RoboDK station: Example 3 - Unload pallet.rdk

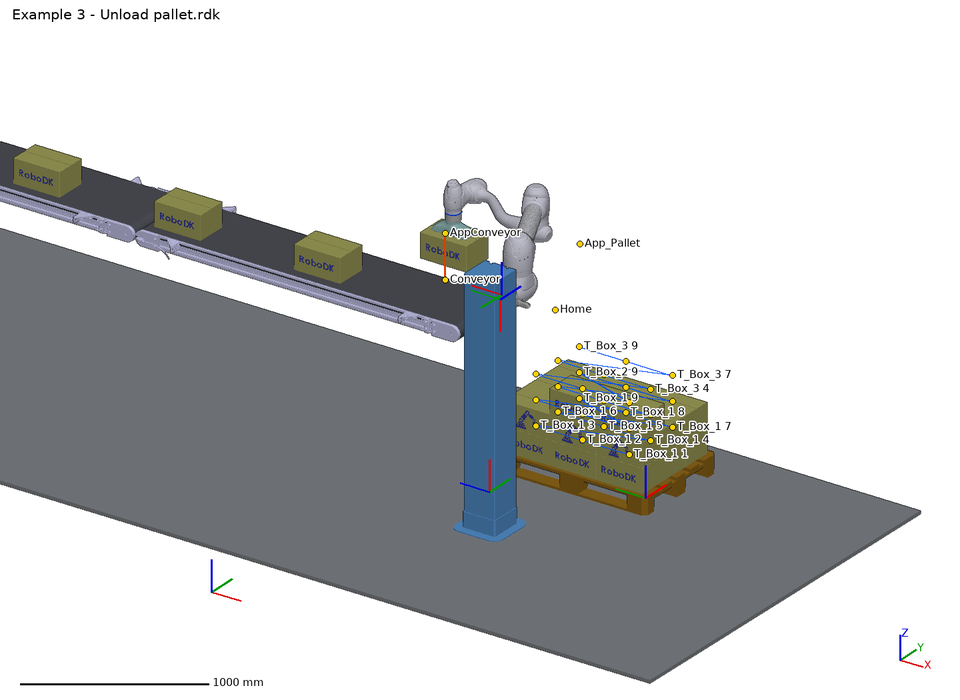
[picture v0: the station drawn from its stored meshes, robots at their saved joint values, targets as dots, program paths as lines]
Station Example 3 - Unload pallet. Poses are relative to the parent item; angles as X-Y-Z fixed-axis rotations.
  - frame Linear Rail Base at (750, 1500, 200) mm, rotated rx 0 ry -90 rz 0 deg
    - robot Linear Rail: 1 axes
        modified DH rows (alpha deg, a mm, theta deg, d mm): 0, 0, 0, 0 linear
        base shift (0, 0, 0) mm, rotated rx 0 ry 90 rz 0 deg
        joint limits [0] to [1200]; home [0]; saved at [1095.81]
      - frame Doosan Robotics M1013 Base at (0, 100, 0) mm, rotated rx 90 ry 0 rz 180 deg
        - robot Doosan Robotics M1013: 6 axes, payload 10 kg, reach 1300 mm, repeatability 0.1 mm, weight 33 kg
            modified DH rows (alpha deg, a mm, theta deg, d mm): 0, 0, 0, 152.5; -90, 0, -90, 34.506; 0, 620, -90, 0; -90, 0, 0, 559; 90, 0, 0, 0; -90, 0, 180, 121
            base shift (0, 0, 0) mm, rotated rx 0 ry 0 rz 180 deg
            joint limits [-120, -100, -160, -360, -360, -360] to [-60, 100, 160, 360, 360, 360]; home [0, 0, -90, 0, 0, 0]; saved at [-88.555, 26.122, 60.089, 89.791, -91.38, -93.79]
          - tool Tool, TCP at (0, 0, 69) mm, size 225 x 100 x 69 mm, geometry from Tool.step
            - object Box_3 3 at (5, 0, 77.5) mm, rotated rx 180 ry 0 rz -90 deg, size 300 x 202 x 153 mm, geometry from Box.step
  - frame Conveyor Belt Base at (57.17, 2600, 730) mm, rotated rx 0 ry 0 rz -180 deg
    - robot Conveyor Belt: 1 axes
        modified DH rows (alpha deg, a mm, theta deg, d mm): 0, 0, 0, 0 linear
        base shift (0, 0, 0) mm, rotated rx 0 ry 90 rz 0 deg
        joint limits [-500000] to [500000]; home [0]; saved at [-494045.004]
      - frame Conveyor at (0, 0, 0) mm
        - object Box_3 9 at (499511.41, 284.96, 74.77) mm, rotated rx 0.03 ry -0.02 rz -90.02 deg, size 300 x 202 x 153 mm, geometry from Box.step
        - object Box_3 8 at (498601.41, 284.96, 74.77) mm, rotated rx 0.03 ry -0.02 rz -90.02 deg, size 300 x 202 x 153 mm, geometry from Box.step
        - object Box_3 7 at (497699.41, 284.96, 74.77) mm, rotated rx 0.03 ry -0.02 rz -90.02 deg, size 300 x 202 x 153 mm, geometry from Box.step
        - object Box_3 6 at (496784.41, 284.96, 74.77) mm, rotated rx 0.03 ry -0.02 rz -90.02 deg, size 300 x 202 x 153 mm, geometry from Box.step
        - object Box_3 5 at (495873.41, 284.96, 74.77) mm, rotated rx 0.03 ry -0.02 rz -90.02 deg, size 300 x 202 x 153 mm, geometry from Box.step
        - object Box_3 4 at (494970.41, 284.96, 74.77) mm, rotated rx 0.03 ry -0.02 rz -90.02 deg, size 300 x 202 x 153 mm, geometry from Box.step
    - target AppConveyor (Cartesian target) at (166.39, 285.12, 428.8) mm, rotated rx -179.99 ry 0.02 rz 179.99 deg; joints [-88.768, 29.095, 58.796, 89.941, -91.212, -92.104, 1095.81] of Doosan Robotics M1013
    - target Conveyor (Cartesian target) at (166.37, 284.98, 152.27) mm, rotated rx -179.98 ry 0.03 rz 179.98 deg; joints [-88.76, 29.09, 58.79, 89.94, -91.21, -92.1, 819.16] of Doosan Robotics M1013
    - object Conveyor at (2400, 440, -50) mm, rotated rx 0 ry 0 rz -90 deg, size 597 x 2090.8 x 107.2 mm
    - object Conveyor at (4500, 440, -50) mm, rotated rx 0 ry 0 rz -90 deg, size 597 x 2090.8 x 107.2 mm
  - frame Pallet at (1350, 2080, 100) mm, rotated rx 0 ry 0 rz 90 deg
    - object Pallet at (-0.19, 0.17, 1.21) mm, size 660 x 990 x 118.8 mm, geometry from User Library-Europallet.igs
    - target T_Box_1 1 (Cartesian target) at (120, 190, 157.5) mm, rotated rx -180 ry 0 rz -90 deg; joints [-92.925, -96.78, 118.114, 92.725, -88.936, -158.691, 192] of Doosan Robotics M1013
    - target T_Box_1 2 (Cartesian target) at (120, 490, 157.5) mm, rotated rx 180 ry 0 rz -90 deg; joints [-100.509, -74.899, 134.13, 95.421, -80.984, -121.197, 192] of Doosan Robotics M1013
    - target T_Box_1 3 (Cartesian target) at (120, 790, 157.5) mm, rotated rx 180 ry 0 rz -90 deg; joints [-83.756, -35.637, 131.426, 90.632, -96.212, -84.176, 192] of Doosan Robotics M1013
    - target T_Box_1 4 (Cartesian target) at (320, 190, 157.5) mm, rotated rx -180 ry 0 rz -90 deg; joints [-92.925, -78.491, 98.933, 92.741, -88.979, -159.582, 192] of Doosan Robotics M1013
    - target T_Box_1 5 (Cartesian target) at (320, 490, 157.5) mm, rotated rx -180 ry 0 rz -90 deg; joints [-100.509, -62.114, 112.355, 96.766, -81.94, -130.236, 192] of Doosan Robotics M1013
    - target T_Box_1 6 (Cartesian target) at (320, 790, 157.5) mm, rotated rx 180 ry 0 rz -90 deg; joints [-83.756, -34.116, 110.225, 88.495, -96.061, -103.971, 192] of Doosan Robotics M1013
    - target T_Box_1 7 (Cartesian target) at (520, 190, 157.5) mm, rotated rx 180 ry 0 rz -90 deg; joints [-92.925, -60.698, 73.974, 92.847, -89.329, -166.74, 192] of Doosan Robotics M1013
    - target T_Box_1 8 (Cartesian target) at (520, 490, 157.5) mm, rotated rx 180 ry 0 rz -90 deg; joints [-100.509, -48.668, 87.076, 98.271, -83.494, -142.063, 192] of Doosan Robotics M1013
    - target T_Box_1 9 (Cartesian target) at (520, 790, 157.5) mm, rotated rx 180 ry 0 rz -90 deg; joints [-83.756, -26.873, 85.087, 86.702, -95.305, -121.939, 192] of Doosan Robotics M1013
    - target T_Box_2 1 (Cartesian target) at (120, 190, 310) mm, rotated rx -180 ry 0 rz -90 deg; joints [-100, -10.355, 75.202, 134.117, -34.001, -139.471, 347.5] of Doosan Robotics M1013
    - target T_Box_2 2 (Cartesian target) at (120, 490, 310) mm, rotated rx 180 ry 0 rz -90 deg; joints [-100, -10.355, 75.202, 134.117, -34.001, -139.471, 347.5] of Doosan Robotics M1013
    - target T_Box_2 3 (Cartesian target) at (120, 790, 310) mm, rotated rx 180 ry 0 rz -90 deg; joints [-100, -10.355, 75.202, 134.117, -34.001, -139.471, 347.5] of Doosan Robotics M1013
    - target T_Box_2 4 (Cartesian target) at (320, 190, 310) mm, rotated rx -180 ry 0 rz -90 deg; joints [-100, -10.355, 75.202, 134.117, -34.001, -139.471, 347.5] of Doosan Robotics M1013
    - target T_Box_2 5 (Cartesian target) at (320, 490, 310) mm, rotated rx -180 ry 0 rz -90 deg; joints [-100, -10.355, 75.202, 134.117, -34.001, -139.471, 347.5] of Doosan Robotics M1013
    - target T_Box_2 6 (Cartesian target) at (320, 790, 310) mm, rotated rx 180 ry 0 rz -90 deg; joints [-100, -10.355, 75.202, 134.117, -34.001, -139.471, 347.5] of Doosan Robotics M1013
    - target T_Box_2 7 (Cartesian target) at (520, 190, 310) mm, rotated rx 180 ry 0 rz -90 deg; joints [-100, -10.355, 75.202, 134.117, -34.001, -139.471, 347.5] of Doosan Robotics M1013
    - target T_Box_2 8 (Cartesian target) at (520, 490, 310) mm, rotated rx 180 ry 0 rz -90 deg; joints [-100, -10.355, 75.202, 134.117, -34.001, -139.471, 347.5] of Doosan Robotics M1013
    - target T_Box_2 9 (Cartesian target) at (520, 790, 310) mm, rotated rx 180 ry 0 rz -90 deg; joints [-100, -10.355, 75.202, 134.117, -34.001, -139.471, 347.5] of Doosan Robotics M1013
    - target T_Box_3 1 (Cartesian target) at (120, 190, 462.5) mm, rotated rx -180 ry 0 rz -90 deg; joints [-92.508, -96.765, 118.144, 92.336, -89.086, -158.639, 500] of Doosan Robotics M1013
    - target T_Box_3 2 (Cartesian target) at (120, 490, 462.5) mm, rotated rx 180 ry 0 rz -90 deg; joints [-99.069, -74.746, 134.167, 94.642, -82.201, -120.896, 500] of Doosan Robotics M1013
    - target T_Box_3 3 (Cartesian target) at (120, 790, 462.5) mm, rotated rx 180 ry 0 rz -90 deg; joints [-84.635, -35.739, 131.462, 90.537, -95.338, -84.252, 500] of Doosan Robotics M1013
    - target T_Box_3 4 (Cartesian target) at (320, 190, 462.5) mm, rotated rx -180 ry 0 rz -90 deg; joints [-92.508, -78.478, 98.96, 92.35, -89.123, -159.536, 500] of Doosan Robotics M1013
    - target T_Box_3 5 (Cartesian target) at (320, 490, 462.5) mm, rotated rx -180 ry 0 rz -90 deg; joints [-99.069, -62.008, 112.384, 95.812, -83.027, -129.979, 500] of Doosan Robotics M1013
    - target T_Box_3 6 (Cartesian target) at (320, 790, 462.5) mm, rotated rx 180 ry 0 rz -90 deg; joints [-84.635, -34.196, 110.254, 88.704, -95.206, -104.001, 500] of Doosan Robotics M1013
    - target T_Box_3 7 (Cartesian target) at (520, 190, 462.5) mm, rotated rx 180 ry 0 rz -90 deg; joints [-92.508, -60.689, 74.002, 92.441, -89.423, -166.699, 500] of Doosan Robotics M1013
    - target T_Box_3 8 (Cartesian target) at (520, 490, 462.5) mm, rotated rx 180 ry 0 rz -90 deg; joints [-99.069, -48.589, 87.102, 97.119, -84.367, -141.837, 500] of Doosan Robotics M1013
    - target T_Box_3 9 (Cartesian target) at (520, 790, 462.5) mm, rotated rx 180 ry 0 rz -90 deg; joints [-100, -10.355, 75.202, 134.117, -34.001, -139.471, 500] of Doosan Robotics M1013
    - target App_Pallet (Cartesian target) at (536.24, 799.31, 1058.38) mm, rotated rx -179.99 ry 0.02 rz -90.01 deg; joints [-84.86, -25.42, 82.51, 87.2, -94.29, -123.01, 1095.81] of Doosan Robotics M1013
    - object Box_1 1 at (120, 185, 80) mm, size 300 x 202 x 153 mm, geometry from Box.step
    - object Box_1 2 at (120, 485, 80) mm, size 300 x 202 x 153 mm, geometry from Box.step
    - object Box_1 3 at (120, 785, 80) mm, size 300 x 202 x 153 mm, geometry from Box.step
    - object Box_1 4 at (320, 185, 80) mm, size 300 x 202 x 153 mm, geometry from Box.step
    - object Box_1 5 at (320, 485, 80) mm, size 300 x 202 x 153 mm, geometry from Box.step
    - object Box_1 6 at (320, 785, 80) mm, size 300 x 202 x 153 mm, geometry from Box.step
    - object Box_1 7 at (520, 185, 80) mm, size 300 x 202 x 153 mm, geometry from Box.step
    - object Box_1 8 at (520, 485, 80) mm, size 300 x 202 x 153 mm, geometry from Box.step
    - object Box_1 9 at (520, 785, 80) mm, size 300 x 202 x 153 mm, geometry from Box.step
    - object Box_2 1 at (520, 785, 232.5) mm, rotated rx 0 ry 0 rz -180 deg, size 300 x 202 x 153 mm, geometry from Box.step
    - object Box_2 2 at (520, 485, 232.5) mm, rotated rx 0 ry 0 rz -180 deg, size 300 x 202 x 153 mm, geometry from Box.step
    - object Box_2 3 at (520, 185, 232.5) mm, rotated rx 0 ry 0 rz -180 deg, size 300 x 202 x 153 mm, geometry from Box.step
    - object Box_2 4 at (320, 785, 232.5) mm, rotated rx 0 ry 0 rz -180 deg, size 300 x 202 x 153 mm, geometry from Box.step
    - object Box_2 5 at (320, 485, 232.5) mm, rotated rx 0 ry 0 rz -180 deg, size 300 x 202 x 153 mm, geometry from Box.step
    - object Box_2 6 at (320, 185, 232.5) mm, rotated rx 0 ry 0 rz -180 deg, size 300 x 202 x 153 mm, geometry from Box.step
    - object Box_2 7 at (120, 785, 232.5) mm, rotated rx 0 ry 0 rz -180 deg, size 300 x 202 x 153 mm, geometry from Box.step
    - object Box_2 8 at (120, 485, 232.5) mm, rotated rx 0 ry 0 rz -180 deg, size 300 x 202 x 153 mm, geometry from Box.step
    - object Box_2 9 at (120, 185, 232.5) mm, rotated rx 0 ry 0 rz -180 deg, size 300 x 202 x 153 mm, geometry from Box.step
    - object Box_3 1 at (120, 185, 385) mm, size 300 x 202 x 153 mm, geometry from Box.step
    - object Box_3 2 at (120, 485, 385) mm, size 300 x 202 x 153 mm, geometry from Box.step
  - frame World at (0, 0, 0) mm
    - target Home (joint target) at (876.47, 1924.34, 1140.31) mm, rotated rx -180 ry 0 rz 0 deg; joints [-90, -100, 160, 90, -90, -120, 1095.8] of Doosan Robotics M1013
    - target ConvHome (Cartesian target) at (500057.17, 2600, 730) mm, rotated rx 0 ry 0 rz -180 deg; joints [-500000, 0, 0, 0, 0, 0, 0] of Conveyor Belt
    - target ConvRun (Cartesian target) at (392.51, 2433.37, 999.75) mm, rotated rx 180 ry 0 rz 2.38 deg; joints [50000, -58.983, -101.068, -19.936, -5.281, -2.394, 1150.26] of Conveyor Belt
    - object Floor at (-7500, 480, -30) mm, size 10000 x 2500 x 20 mm, geometry from Floor.step
  - program ReplaceObjects (1 instructions, listed below)
  - program MainProgram (167 instructions, listed below)
  - program AppPallet (3 instructions, listed below)
  - program DropConveyor (6 instructions, listed below)
  - program GoHome (3 instructions, listed below)
  - program Pick (1 instructions, listed below)
  - program RunConveyor (2 instructions, listed below)
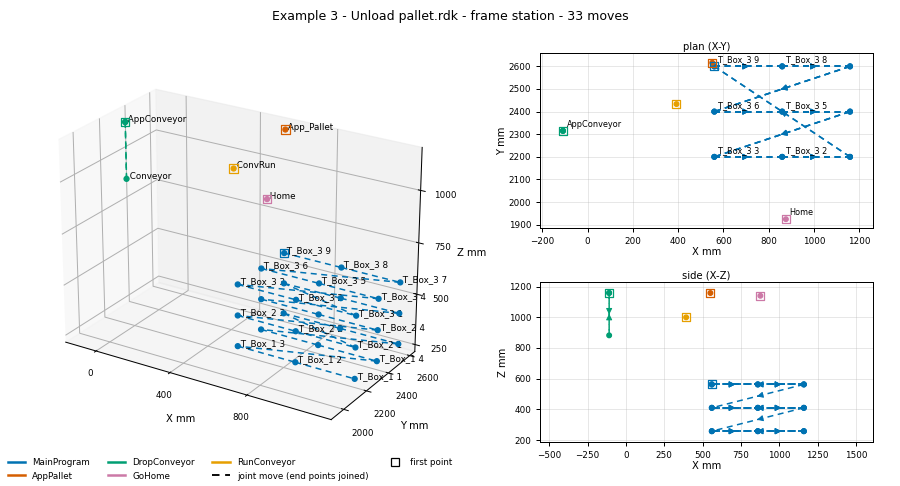
[picture p0: tool path of Example 3 - Unload pallet.rdk in frame station, 33 of 33 moves have a stored position in this frame; points joined in program order, loops and branches not executed]

--- program ReplaceObjects (robot Doosan Robotics M1013) ---
  Replace objects

--- program MainProgram (robot Doosan Robotics M1013) ---
  Call GoHome
  Call ReplaceObjects
  Pause 10.0 s
  Run RunConveyor
  Set Ref.: Pallet
  MoveJ (T_Box_3 9)
  Call Pick
  Call AppPallet
  Call DropConveyor
  Call AppPallet
  Set Ref.: Pallet
  MoveJ (T_Box_3 8)
  Call Pick
  Call AppPallet
  Call DropConveyor
  Call AppPallet
  Set Ref.: Pallet
  MoveJ (T_Box_3 7)
  Call Pick
  Call AppPallet
  Call DropConveyor
  Call AppPallet
  Set Ref.: Pallet
  MoveJ (T_Box_3 6)
  Call Pick
  Call AppPallet
  Call DropConveyor
  Call AppPallet
  Set Ref.: Pallet
  MoveJ (T_Box_3 5)
  Call Pick
  Call AppPallet
  Call DropConveyor
  Call AppPallet
  Set Ref.: Pallet
  MoveJ (T_Box_3 4)
  Call Pick
  Call AppPallet
  Call DropConveyor
  Call AppPallet
  Set Ref.: Pallet
  MoveJ (T_Box_3 3)
  Call Pick
  Call AppPallet
  Call DropConveyor
  Call AppPallet
  Set Ref.: Pallet
  MoveJ (T_Box_3 2)
  Call Pick
  Call AppPallet
  Call DropConveyor
  Call AppPallet
  Set Ref.: Pallet
  MoveJ (T_Box_3 1)
  Call Pick
  Call AppPallet
  Call DropConveyor
  Call AppPallet
  Set Ref.: Pallet
  MoveJ (T_Box_2 9)
  Call Pick
  Call AppPallet
  Call DropConveyor
  Call AppPallet
  Set Ref.: Pallet
  MoveJ (T_Box_2 8)
  Call Pick
  Call AppPallet
  Call DropConveyor
  Call AppPallet
  Set Ref.: Pallet
  MoveJ (T_Box_2 7)
  Call Pick
  Call AppPallet
  Call DropConveyor
  Call AppPallet
  Set Ref.: Pallet
  MoveJ (T_Box_2 6)
  Call Pick
  Call AppPallet
  Call DropConveyor
  Call AppPallet
  Set Ref.: Pallet
  MoveJ (T_Box_2 5)
  Call Pick
  Call AppPallet
  Call DropConveyor
  Call AppPallet
  Set Ref.: Pallet
  MoveJ (T_Box_2 4)
  Call Pick
  Call AppPallet
  Call DropConveyor
  Call AppPallet
  Set Ref.: Pallet
  MoveJ (T_Box_2 3)
  Call Pick
  Call AppPallet
  Call DropConveyor
  Call AppPallet
  Set Ref.: Pallet
  MoveJ (T_Box_2 2)
  Call Pick
  Call AppPallet
  Call DropConveyor
  Call AppPallet
  Set Ref.: Pallet
  MoveJ (T_Box_2 1)
  Call Pick
  Call AppPallet
  Call DropConveyor
  Call AppPallet
  Set Ref.: Pallet
  MoveJ (T_Box_1 9)
  Call Pick
  Call AppPallet
  Call DropConveyor
  Call AppPallet
  Set Ref.: Pallet
  MoveJ (T_Box_1 8)
  Call Pick
  Call AppPallet
  Call DropConveyor
  Call AppPallet
  Set Ref.: Pallet at (-100, 580, -600) mm, rotated rx 90 ry 0 rz 90 deg
  MoveJ (T_Box_1 7)
  Call Pick
  Call AppPallet
  Call DropConveyor
  Call AppPallet
  Set Ref.: Pallet at (-100, 580, -600) mm, rotated rx 90 ry 0 rz 90 deg
  MoveJ (T_Box_1 6)
  Call Pick
  Call AppPallet
  Call DropConveyor
  Call AppPallet
  Set Ref.: Pallet at (-100, 580, -600) mm, rotated rx 90 ry 0 rz 90 deg
  MoveJ (T_Box_1 5)
  Call Pick
  Call AppPallet
  Call DropConveyor
  Call AppPallet
  Set Ref.: Pallet at (-100, 580, -600) mm, rotated rx 90 ry 0 rz 90 deg
  MoveJ (T_Box_1 4)
  Call Pick
  Call AppPallet
  Call DropConveyor
  Call AppPallet
  Set Ref.: Pallet at (-100, 580, -600) mm, rotated rx 90 ry 0 rz 90 deg
  MoveJ (T_Box_1 3)
  Call Pick
  Call AppPallet
  Call DropConveyor
  Call AppPallet
  Set Ref.: Pallet at (-100, 580, -600) mm, rotated rx 90 ry 0 rz 90 deg
  MoveJ (T_Box_1 2)
  Call Pick
  Call AppPallet
  Call DropConveyor
  Call AppPallet
  Set Ref.: Pallet at (-100, 580, -600) mm, rotated rx 90 ry 0 rz 90 deg
  MoveJ (T_Box_1 1)
  Call Pick
  Call AppPallet
  Call DropConveyor
  Call AppPallet
  Call GoHome

--- program AppPallet (robot Doosan Robotics M1013) ---
  Set Ref.: Pallet
  Set Tool: Tool
  MoveJ (App_Pallet)

--- program DropConveyor (robot Doosan Robotics M1013) ---
  Set Ref.: Conveyor Belt Base
  Set Tool: Tool
  MoveJ (AppConveyor)
  MoveJ (Conveyor)
  Detach from Tool
  MoveJ (AppConveyor)

--- program GoHome (robot Doosan Robotics M1013) ---
  Set Ref.: World
  Set Tool: Tool
  MoveJ (Home)

--- program Pick (robot Doosan Robotics M1013) ---
  Attach to Tool

--- program RunConveyor (robot Conveyor Belt) ---
  Set Ref.: World
  MoveJ (ConvRun)
